// TIA Portal V18 export
TYPE "Condition_Check"
// stored: IsFailsafeCompliant false
   STRUCT
      Date_time : DTL;
      Pressure_achieve_time : DInt;
      Leakage_Pressure : Real;
      Status : Int;
   END_STRUCT;
END_TYPE
